FUNCTION_BLOCK FB_PrintModule EXTENDS T_NamedBase
VAR_INPUT
  IbPrinterHood           : BOOL;
  IbServiceDoors          : BOOL;
  IbExhaustVacuumWarning  : BOOL;
  IbExhaustVacuumError    : BOOL;
  IbExhaustFUError        : BOOL;
  IbDriftControlError     : BOOL;
  IbDriftControlMissMarks : BOOL;
  IbSafetyNOk             : BOOL;
END_VAR

VAR
  //config
  _nIdx                   : UDINT;   // for visu selection only (remove later) 
  _pAdsPm                 : POINTER TO ST_ADS_PM; //ads config/status interface
  _fResolutionPrint       : LREAL;
  _fResolutionSubPx       : LREAL;
  _fEncoderResolution     : LREAL;   // encoder resolution for EL5101 (input um/pulse)
  
  // status

  
  // instances
  fbPrintPosition         : FB_PrintPositionDmax;
  
  // helper
  fSpeed, fSpeedMpMin     : LREAL;
  lPos_SubPx, lPos_Px     : DINT;
  fPos_um                 : LREAL;
  
  
  // messaging
  fb_MsgQueue             : FB_MSG_QUEUE;                 (*Message queue*)
  fb_MsgHandler           : FB_MSG_HANDLER;               (*Message handler*)
  sL_MsgConfig            : ST_MSG_CONFIG;                (*Message config*)
  fb_Msg                  : ARRAY [1..iC_NUM_MSG] OF FB_MESSAGE;  (*Messages*)
  
  // view
  
  // testing
  _bSim : BOOL;
END_VAR

VAR CONSTANT
  (*Messaging*)
  iC_NUM_MSG              : INT := 8;
END_VAR



fbPrintPosition();
fSpeed := fbPrintPosition.getSpeed(fSpeedMpMin=>fSpeedMpMin);
lPos_SubPx := fbPrintPosition.getPosition(nPosition_px=>lPos_Px, fPosition_um=>fPos_um);



Messaging();

PROPERTY bSim : BOOL
GET
bSim := _bSim;
END_GET
SET
_bSim := bSim;
END_SET
END_PROPERTY

(*
  Encoder resolution.
*)
PROPERTY fEncoderResolution : LREAL
GET
fEncoderResolution := _fEncoderResolution;
END_GET
SET
_fEncoderResolution := fEncoderResolution;
END_SET
END_PROPERTY

METHOD init : BOOL
VAR_INPUT
  nIdx                : UDINT;                // module id
  pAdsPm              : POINTER TO ST_ADS_PM; // module ads interface

  // config print
  fPrintResolution    : LREAL := 600;         // print(head) resolution in [dpi]
  fSubPxResolution    : LREAL := 32;          // SubPixel resolution [SubPx], resolution factor (fI_PrintResolution*fI_SubPxResolution=>Output resolution)
  fTaskCycleTime      : LREAL;                // Task cycle time in [s]

  nBlockId            : INT;                  // block id for message
END_VAR
VAR CONSTANT
  fC_PROD_MASTER_SPEED                      : LREAL := 5.0;    (*[m/min]*)
END_VAR
IF pAdsPm = 0 THEN
  LogError('Invalid parameter');
  RETURN;
END_IF

// save config
_nIdx := nIdx;
_pAdsPm := pAdsPm;
_fResolutionPrint := fPrintResolution;
_fResolutionSubPx := fSubPxResolution;

// positioning
fbPrintPosition.Init(
  fPrintResolution:=fPrintResolution,
  fSubPxResolution:=fSubPxResolution,
  fTaskCycleTime:=fTaskCycleTime,
  fProdSpeedMpMin:=fC_PROD_MASTER_SPEED
);


(*Messaging*)
sL_MsgConfig.bI_Enable       := TRUE;
sL_MsgConfig.pI_FbMsgHandler := ADR(fb_MsgHandler);
fb_MsgHandler.pI_MsgQueue    := ADR(fb_MsgQueue);
fb_MsgQueue.pI_MsgInterface  := ADR(_pAdsPm^.sO_Message);
fb_MsgQueue.cI_MaxElement    := 6;

(*Messages*)
fb_Msg[1].pI_MsgConfig       := ADR(sL_MsgConfig);
fb_Msg[1].iI_MsgLocation     := nBlockId;
fb_Msg[1].iI_MsgNumber       := eCMa_COVER_INLET;

fb_Msg[2].pI_MsgConfig       := ADR(sL_MsgConfig);
fb_Msg[2].iI_MsgLocation     := nBlockId;
fb_Msg[2].iI_MsgNumber       := eCMa_SECURITY_DOOR_MONITORING;

fb_Msg[3].pI_MsgConfig       := ADR(sL_MsgConfig);
fb_Msg[3].iI_MsgLocation     := nBlockId;
fb_Msg[3].iI_MsgNumber       := eCMa_EXHAUST_SYSTEM_WARNING;

fb_Msg[4].pI_MsgConfig       := ADR(sL_MsgConfig);
fb_Msg[4].iI_MsgLocation     := nBlockId;
fb_Msg[4].iI_MsgNumber       := eCMa_EXHAUST_SYSTEM_ERROR;

fb_Msg[5].pI_MsgConfig       := ADR(sL_MsgConfig);
fb_Msg[5].iI_MsgLocation     := nBlockId;
fb_Msg[5].iI_MsgNumber       := eCMa_EXHAUST_SYSTEM_MALFUNCTION;

fb_Msg[6].pI_MsgConfig       := ADR(sL_MsgConfig);
fb_Msg[6].iI_MsgLocation     := nBlockId;
fb_Msg[6].iI_MsgNumber       := eCMa_DRIFT_CONTR_ERROR;

fb_Msg[7].pI_MsgConfig       := ADR(sL_MsgConfig);
fb_Msg[7].iI_MsgLocation     := nBlockId;
fb_Msg[7].iI_MsgNumber       := eCMa_AXIS_SAFETY_ACCEPTANCE;

fb_Msg[8].pI_MsgConfig       := ADR(sL_MsgConfig);
fb_Msg[8].iI_MsgLocation     := nBlockId;
fb_Msg[8].iI_MsgNumber       := eCPr_SHEET_MARK_DETECTION;
END_METHOD

METHOD Messaging
VAR_INPUT
END_VAR
(*Messaging*)
fb_MsgHandler();

fB_Msg[1](bI_Status := IbPrinterHood);
fB_Msg[2](bI_Status := IbServiceDoors);
fB_Msg[3](bI_Status := IbExhaustVacuumWarning);
fB_Msg[4](bI_Status := IbExhaustVacuumError);
fB_Msg[5](bI_Status := IbExhaustFUError);
fB_Msg[6](bI_Status := IbDriftControlError);
fB_Msg[7](bI_Status := IbSafetyNOk);
fB_Msg[8](bI_Status := IbDriftControlMissMarks);

fb_MsgQueue();
END_METHOD

END_FUNCTION_BLOCK

(* stored: Version 1.1.0.1, ProductVersion 3.1.4024.11
   POU FB_PrintModule: Id {cb9319db-6969-4a30-812e-4f2d714eb08a}, SpecialFunc None
   Folder Position: Id {12a320fc-93c2-445f-a96d-a4cd86407a32}
   Folder Sim: Id {6de8d664-1ecd-4e7c-9e04-bad56ccd972b}
   Property bSim: Id {0f604c0e-9e5d-44dd-b620-672fedba6798}
   Get Get: Id {eed6e031-ccb0-4834-afd4-be86a2055e6a}
   Set Set: Id {0514b0f1-83fc-4960-94d7-be479b9c0ddd}
   Property fEncoderResolution: Id {7b76ff9d-3552-4e96-b7c1-eeed2dc4e44b}
   Get Get: Id {b14c77fd-b6aa-4ec1-9da0-882cd005b6f0}
   Set Set: Id {0ff2555c-4a0e-4ef4-be5a-22cbb71c7c0d}
   Method init: Id {4338a7a6-6293-49ad-a96d-3660b8a91900}
   Method Messaging: Id {643d2082-2a1e-46ab-80d2-9108069a18fe} *)
